// TIA Portal V18 export
DATA_BLOCK "DB_DQ"   // DB3
{ S7_Optimized_Access := 'FALSE' }
VERSION : 0.1
// stored: AutoNumber true, DBAccessibleFromOPCUA true, DBAccessibleFromWebserver true, IsOnlyStoredInLoadMemory false, IsWriteProtectedInAS false
   VAR
      out_BeaconGreen : Bool;
      out_BeaconRed : Bool;
      out_BeaconYellow : Bool;
      out_GenPallet : Bool;
      out_GenBox : Bool;
      out_5 : Bool;
      out_6 : Bool;
      out_7 : Bool;
      out_8 : Bool;
      out_Cov_0 : Bool;
      out_Cov_1 : Bool;
      out_Cov_2 : Bool;
      out_Cov_3 : Bool;
      out_Cov_4 : Bool;
      out_Cov_5 : Bool;
      out_15 : Bool;
      out_Picker : Bool;
      out_17 : Bool;
      out_18 : Bool;
      out_19 : Bool;
      out_20 : Bool;
      out_21 : Bool;
      out_22 : Bool;
      out_23 : Bool;
      out_BladesForward : Bool;
      out_BladesBackward : Bool;
      out_26 : Bool;
      out_27 : Bool;
      out_28 : Bool;
      out_29 : Bool;
      out_30 : Bool;
      out_31 : Bool;
   END_VAR
BEGIN
END_DATA_BLOCK
